FUNCTION_BLOCK SLEEP (* Service Interface Function Block Type *)
  (* Standard: 61499-1 Annex A; Description: Copyright (c) 2017 fortiss GmbH This program and the accompanying materials are made available under the terms of the Eclipse Public License 2.0 which is available at https://www.eclipse.org/legal/epl-2.0/ SPDX-License-Identifier: EPL-2.0 *)
  (* Version 1.0, 2017-09-21, Alois Zoitl, fortiss GmbH, initial API and implementation and/or initial documentation *)
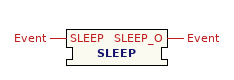
  EVENT_INPUT
    SLEEP;
  END_EVENT
  EVENT_OUTPUT
    SLEEP_O;
  END_EVENT
END_FUNCTION_BLOCK
